(* PLC project Senza_nome, Sconosciuto Senza_nome 1 *)
(* stored: creationDateTime 2026-08-24T11:36:29, modificationDateTime 2026-08-24T12:03:28 *)

PROGRAM program0
  VAR
    s1 AT %IX100.0 : BOOL;
    s2 AT %IX100.1 : BOOL;
    s3 AT %IX100.2 : BOOL;
    K1 AT %QX100.0 : BOOL;
    K2 AT %QX100.1 : BOOL;
    LDP AT %QX100.2 : BOOL;
  END_VAR

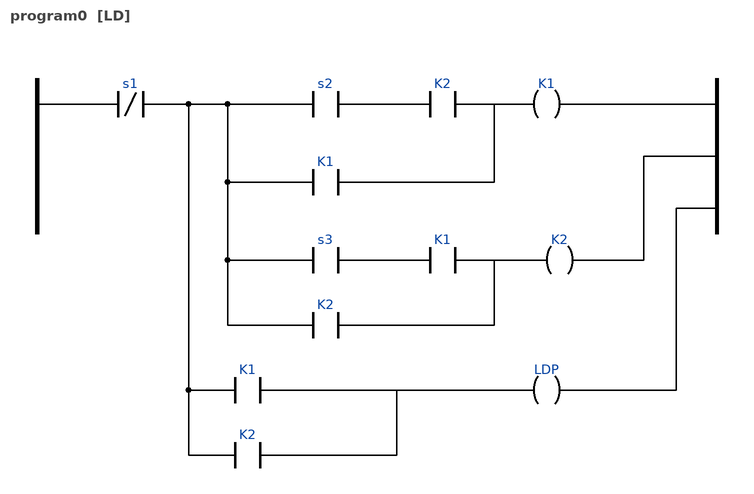
(* LD diagram, written out as Structured Text *)
K1 := NOT s1 AND (s2 AND K2 OR K1);
K2 := NOT s1 AND (s3 AND K1 OR K2);
LDP := NOT s1 AND (K1 OR K2);
END_PROGRAM

CONFIGURATION Config0
  RESOURCE Res0 ON PLC
    TASK task0(INTERVAL := T#20ms, PRIORITY := 0);
    PROGRAM instance0 WITH task0 : program0;
  END_RESOURCE
END_CONFIGURATION
